// CODESYS_Control_for_Raspberry_Pi/Application/visualization/ups_s2/ups_s2_state
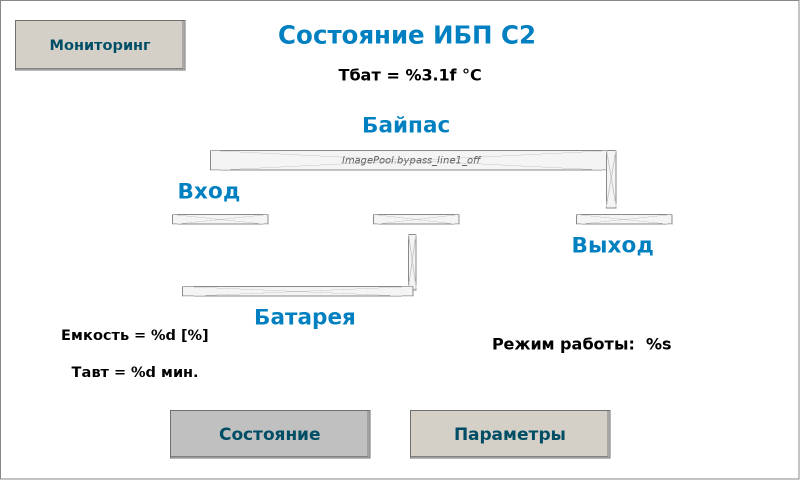
VISUALIZATION ups_s2_state  // 800x480, background image ImagePool.mpx_state_bg
    Rectangle (204,20 406x30), "Состояние ИБП С2"
    Button (410,410 200x48), "Параметры"
        OnMouseClick:  Assign=ups_s2_params, Type=Assignment
    Button (170,410 200x48), "Состояние", pressed state: PLC_PRG.var_true
    Rectangle (350,110 112x30), "Байпас"
    Rectangle (246,302 118x30), "Батарея"
    Rectangle (166,176 86x30), "Вход"
    Rectangle (560,230 106x30), "Выход"
    Rectangle (30,320 210x30), "Емкость = %d [%]", text variable: PLC_PRG.ips_s2_battery_capacity
    Rectangle (30,357 210x30), "Tавт = %d мин.", text variable: PLC_PRG.ips_s2_time_m
    Image (210,150 402x20), image: ImagePool.bypass_line1_off
        p84334746: PLC_PRG.ips_s2_bypass_line_state
    Image (606,150 10x58), image: ImagePool.bypass_arrow_off
        p84334746: PLC_PRG.ips_s2_bypass_arrow_state
    Image (576,214 96x10), image: ImagePool.arrow_off
        p84334746: PLC_PRG.ips_s2_output_state
    Image (172,214 96x10), image: ImagePool.arrow_off
        p84334746: PLC_PRG.ips_s2_input_state
    Image (408,234 8x56), image: ImagePool.battery_arrow_off
        p84334746: PLC_PRG.ips_s2_battery_arrow_state
    Image (182,286 231x10), image: ImagePool.battery_line_off
        p84334746: PLC_PRG.ips_s2_battery_line_state
    Button (15,20 170x50), "Мониторинг"
        OnMouseClick:  Assign=monitoring, Type=Assignment
    Rectangle (372,212 85x14)
    Image (373,214 86x10), image: ImagePool.arrow_off
        p84334746: PLC_PRG.ips_s2_arrow_state
    Rectangle (280,60 260x30), "Tбат = %3.1f °С", text variable: PLC_PRG.ips_s2_temp_real
    Rectangle (396,329 372x30), "Режим работы: %s", text variable: PLC_PRG.mpx_s2_state_string
    hotkey  Id=481037385728, Key=KeyDown=True, KeyName=0, VisuElemId=38
    hotkey  Id=481038434304, Key=KeyName=0, VisuElemId=38
END_VISUALIZATION

// CODESYS_Control_for_Raspberry_Pi/Application/visualization/main
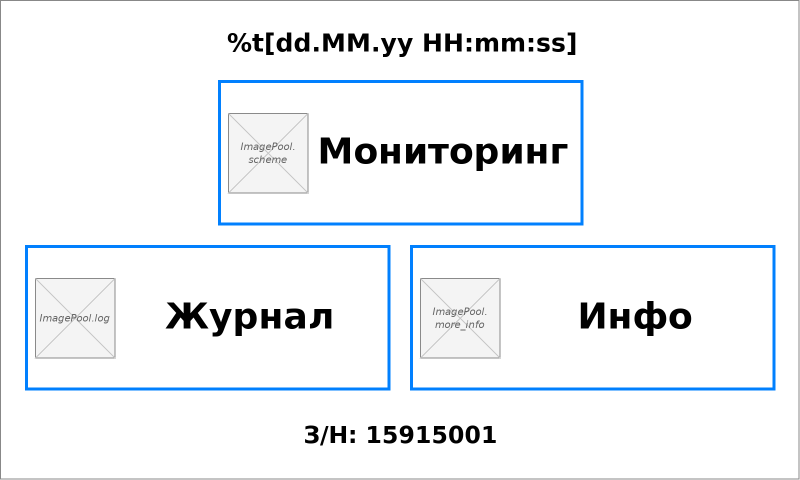
VISUALIZATION main  // 800x480, background image ImagePool.bg_800
    Group (218,80 365x145)
        OnMouseClick:  Assign=monitoring, Type=Assignment
        RoundedRectangle (0,0 365x145)
            OnMouseClick:  Assign=ups_s2_state, Type=Assignment
        RoundedRectangle (95,43 260x56), "Мониторинг"
        Image (10,33 80x80), image: ImagePool.scheme
    Group (25,245 365x145)
        OnMouseClick:  Assign=logs, Type=Assignment
        RoundedRectangle (0,0 365x145)
            OnMouseClick:  Assign=ups_s2_state, Type=Assignment
        RoundedRectangle (95,43 260x56), "Журнал"
            OnMouseClick:  Assign=ups_s2_state, Type=Assignment
        Image (10,33 80x80), image: ImagePool.log
    Group (410,245 365x145)
        OnMouseClick:  Assign=more, Type=Assignment
        RoundedRectangle (0,0 365x145)
            OnMouseClick:  Assign=ups_s2_state, Type=Assignment
        RoundedRectangle (95,43 260x56), "Инфо"
        Image (10,33 80x80), image: ImagePool.more_info
    Rectangle (215,20 375x45), "%t[dd.MM.yy HH:mm:ss]"
    Label (303,420 195x30), "З/Н: 15915001"
END_VISUALIZATION

// CODESYS_Control_for_Raspberry_Pi/Application/visualization/info
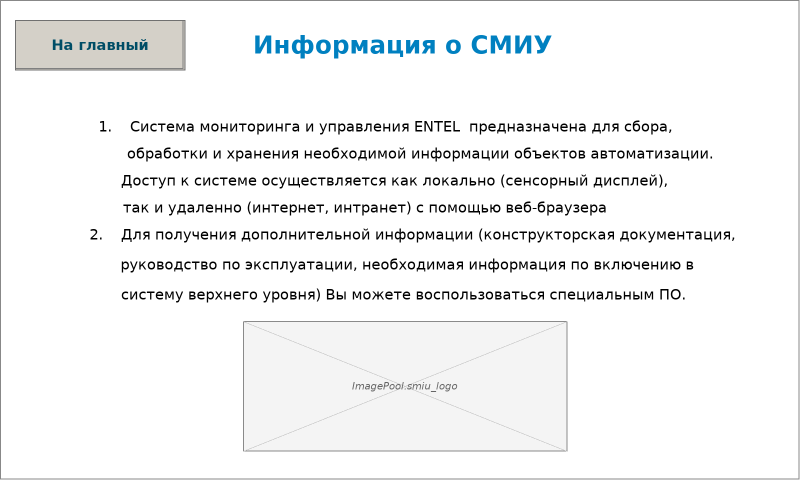
VISUALIZATION info  // 800x480, background image ImagePool.bg_800
    Rectangle (200,30 406x30), "Информация о СМИУ"
    Button (15,20 170x50), "На главный"
        OnMouseClick:  Assign=main, Type=Assignment
    Label (78,108 615x37), "1. Система мониторинга и управления ENTEL предназначена для сбора,"
    Label (120,135 601x37), "обработки и хранения необходимой информации объектов автоматизации."
    Label (99,162 591x37), "Доступ к системе осуществляется как локально (сенсорный дисплей),"
    Label (42,189 646x37), "так и удаленно (интернет, интранет) с помощью веб-браузера"
    Label (105,216 615x37), "2. Для получения дополнительной информации (конструкторская документация,"
    Label (120,243 601x37)
    Label (114,246 591x37), "руководство по эксплуатации, необходимая информация по включению в"
    Label (108,276 591x37), "систему верхнего уровня) Вы можете воспользоваться специальным ПО."
    Image (243,321 324x130), image: ImagePool.smiu_logo
END_VISUALIZATION

// CODESYS_Control_for_Raspberry_Pi/Application/visualization/climate
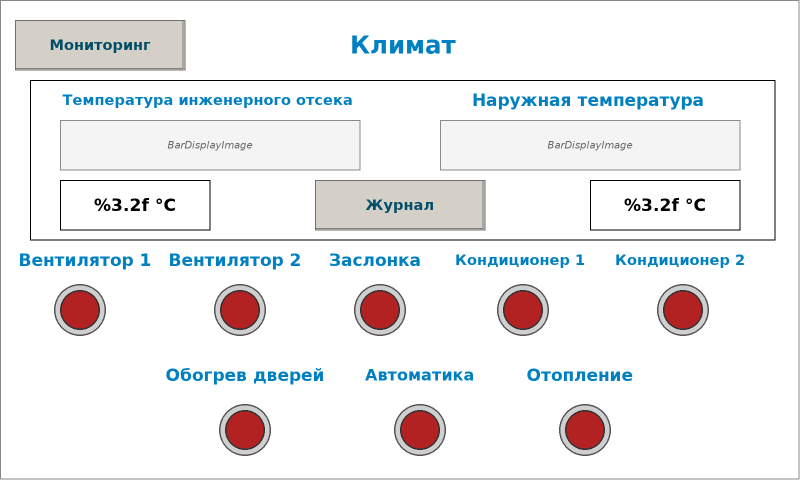
VISUALIZATION climate  // 800x480, background image ImagePool.bg_800
    Rectangle (200,30 406x30), "Климат"
    Button (15,20 170x50), "Мониторинг"
        OnMouseClick:  Assign=monitoring, Type=Assignment
    Rectangle (30,80 745x160)
    Rectangle (35,85 346x30), "Температура инженерного отсека"
    Rectangle (60,180 150x50), "%3.2f °С", text variable: PLC_PRG.climate_temp_in_real
    BarDisplayImage (60,120 300x50), value: PLC_PRG.climate_temp_in_real, style: BarDisplayImage-Gray, scale format: %.1f, scale -10..50
    Rectangle (415,85 346x30), "Наружная температура"
    Rectangle (590,180 150x50), "%3.2f °С", text variable: PLC_PRG.climate_temp_out_real
    BarDisplayImage (440,120 300x50), value: PLC_PRG.climate_temp_out_real, style: BarDisplayImage-Gray, scale format: %.1f, scale -60..80
    Rectangle (345,360 150x30), "Автоматика"
    Lamp1 (390,400 60x60), variable: PLC_PRG.climate_auto_state, style: Lamp-Lamp1-Red
    Lamp1 (50,280 60x60), variable: PLC_PRG.climate_vent_1_state, style: Lamp-Lamp1-Red
    Rectangle (10,250 150x20), "Вентилятор 1"
    Lamp1 (350,280 60x60), variable: PLC_PRG.climate_zaslonka_state, style: Lamp-Lamp1-Red
    Rectangle (320,250 110x20), "Заслонка"
    Rectangle (440,250 160x20), "Кондиционер 1"
    Lamp1 (490,280 66x60), variable: PLC_PRG.climate_condition_1_state, style: Lamp-Lamp1-Red
    Lamp1 (555,400 60x60), variable: PLC_PRG.climate_heat_state, style: Lamp-Lamp1-Red
    Rectangle (505,365 150x20), "Отопление"
    Lamp1 (210,280 60x60), variable: PLC_PRG.climate_vent_2_state, style: Lamp-Lamp1-Red
    Rectangle (160,250 150x20), "Вентилятор 2"
    Rectangle (600,250 160x20), "Кондиционер 2"
    Lamp1 (650,280 66x60), variable: PLC_PRG.climate_condition_2_state, style: Lamp-Lamp1-Red
    Lamp1 (215,400 60x60), variable: PLC_PRG.climate_heat_door_state, style: Lamp-Lamp1-Red
    Rectangle (155,365 180x20), "Обогрев дверей"
    Button (315,180 170x50), "Журнал"
        OnMouseClick:  Assign=climate_log, Type=Assignment
    hotkey  Id=481037385728, Key=KeyDown=True, KeyName=0, VisuElemId=3
    hotkey  Id=481038434304, Key=KeyName=0, VisuElemId=3
    hotkey  Id=481037385728, Key=KeyDown=True, KeyName=0, VisuElemId=73
    hotkey  Id=481038434304, Key=KeyName=0, VisuElemId=73
END_VISUALIZATION

// CODESYS_Control_for_Raspberry_Pi/Application/visualization/alarm
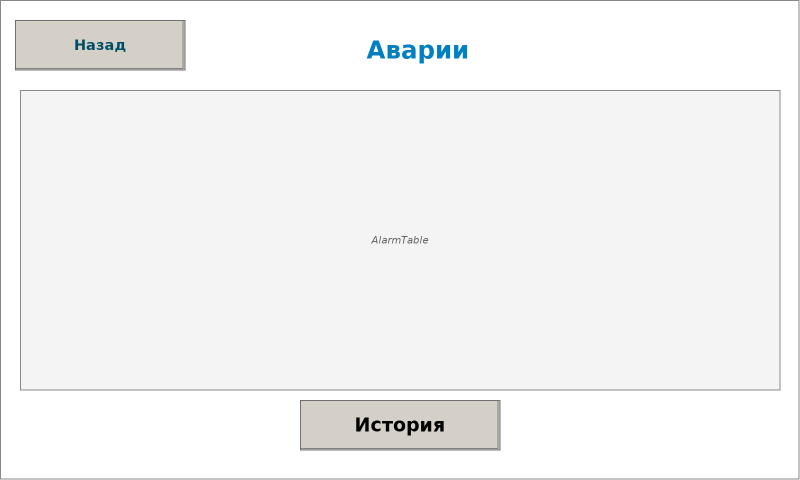
VISUALIZATION alarm  // 800x480, background image ImagePool.bg_800
    Button (300,400 200x50), "История", colour toggle: PLC_PRG.history
        toggle PLC_PRG.history
    Button (15,20 170x50), "Назад"
        OnMouseClick:  Assign=monitoring, Type=Previous
    AlarmTable (20,90 760x300)
        Column[0]: ColumnTitle=Временная отметка
        Column[1]: ColumnTitle=Сообщение
        p1521930926: AlarmGroup
        p1663851261: __All
        p3266827225: PLC_PRG.history
    Rectangle (215,35 406x30), "Аварии"
    hotkey  Id=481037385728, Key=KeyDown=True, KeyName=0, VisuElemId=6
    hotkey  Id=481038434304, Key=KeyName=0, VisuElemId=6
END_VISUALIZATION

// CODESYS_Control_for_Raspberry_Pi/Application/visualization/schrps
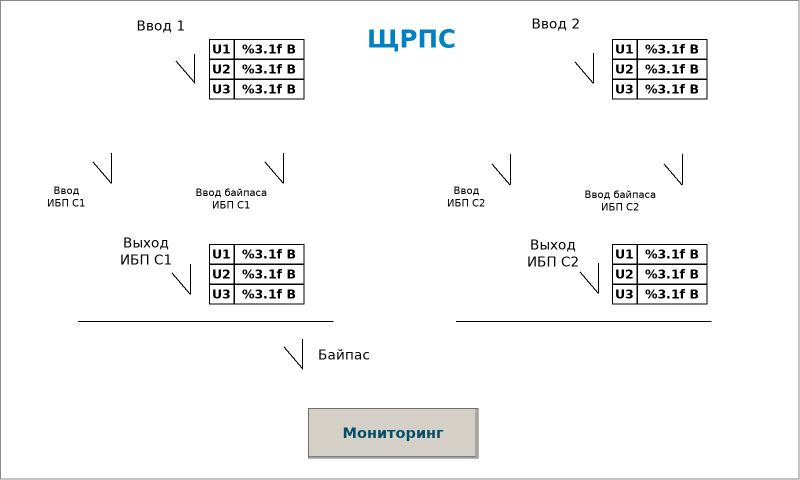
VISUALIZATION schrps  // 800x480, background image ImagePool.shrps
    Button (308,408 170x50), "Мониторинг"
        OnMouseClick:  Assign=monitoring, Type=Assignment
    Rectangle (316,24 191x30), "ЩРПC"
    Line (194,82) (176,61), invisible if: PLC_PRG.shrps_in_1
    Line (111,183) (93,162), invisible if: PLC_PRG.shrps_ups_in_1
    Line (283,183) (265,162), invisible if: PLC_PRG.shrps_bypass_in_1
    Line (190,294) (172,273), invisible if: PLC_PRG.shrps_ups_out_1
    Line (302,368) (284,347), invisible if: PLC_PRG.shrps_bypass_out
    Line (598,293) (580,272), invisible if: PLC_PRG.shrps_ups_out_2
    Line (510,185) (492,164), invisible if: PLC_PRG.shrps_ups_in_2
    Line (682,185) (664,164), invisible if: PLC_PRG.shrps_bypass_in_2
    Line (593,83) (575,62), invisible if: PLC_PRG.shrps_in_2
    Line (194,54) (194,83), invisible if: NOT(PLC_PRG.shrps_in_1)
    Line (283,153) (283,183), invisible if: NOT(PLC_PRG.shrps_bypass_in_1)
    Line (111,153) (111,183), invisible if: NOT(PLC_PRG.shrps_ups_in_1)
    Line (190,264) (190,294), invisible if: NOT(PLC_PRG.shrps_ups_out_1)
    Line (302,339) (302,369), invisible if: NOT(PLC_PRG.shrps_bypass_out)
    Line (598,263) (598,293), invisible if: NOT(PLC_PRG.shrps_ups_out_2)
    Line (682,154) (682,184), invisible if: NOT(PLC_PRG.shrps_bypass_in_2)
    Line (510,154) (510,184), invisible if: NOT(PLC_PRG.shrps_ups_in_2)
    Line (593,53) (593,83), invisible if: NOT(PLC_PRG.shrps_in_2)
    Label (317,340 54x30), "Байпас"
    Label (134,11 54x30), "Ввод 1"
    Label (529,9 54x30), "Ввод 2"
    Label (16,178 101x38), "Ввод ИБП С1"
    Label (416,178 101x38), "Ввод ИБП С2"
    Label (181,180 101x38), "Ввод байпаса ИБП С1"
    Label (570,182 101x38), "Ввод байпаса ИБП С2"
    Group (209,244 95x60)
        Rectangle (25,0 70x20), "%3.1f В", text variable: PLC_PRG.shrps_voltage_3_line_1
        Rectangle (0,0 25x20), "U1"
        Rectangle (0,20 25x20), "U2"
        Rectangle (25,20 70x20), "%3.1f В", text variable: PLC_PRG.shrps_voltage_3_line_2
        Rectangle (0,40 25x20), "U3"
        Rectangle (25,40 70x20), "%3.1f В", text variable: PLC_PRG.shrps_voltage_3_line_3
    Label (112,232 68x39), "Выход ИБП С1"
    Line (456,321) (711,321), colour toggle: PLC_PRG.shrps_ups_bus_2
    Line (78,321) (333,321), colour toggle: PLC_PRG.shrps_ups_bus_1
    Label (519,234 68x39), "Выход ИБП С2"
    Group (209,39 95x60)
        Rectangle (25,0 70x20), "%3.1f В", text variable: PLC_PRG.shrps_voltage_1_line_1
        Rectangle (0,0 25x20), "U1"
        Rectangle (0,20 25x20), "U2"
        Rectangle (25,20 70x20), "%3.1f В", text variable: PLC_PRG.shrps_voltage_1_line_2
        Rectangle (0,40 25x20), "U3"
        Rectangle (25,40 70x20), "%3.1f В", text variable: PLC_PRG.shrps_voltage_1_line_3
    Group (612,39 95x60)
        Rectangle (25,0 70x20), "%3.1f В", text variable: PLC_PRG.shrps_voltage_2_line_1
        Rectangle (0,0 25x20), "U1"
        Rectangle (0,20 25x20), "U2"
        Rectangle (25,20 70x20), "%3.1f В", text variable: PLC_PRG.shrps_voltage_2_line_2
        Rectangle (0,40 25x20), "U3"
        Rectangle (25,40 70x20), "%3.1f В", text variable: PLC_PRG.shrps_voltage_2_line_3
    Group (612,244 95x60)
        Rectangle (25,0 70x20), "%3.1f В", text variable: PLC_PRG.shrps_voltage_4_line_1
        Rectangle (0,0 25x20), "U1"
        Rectangle (0,20 25x20), "U2"
        Rectangle (25,20 70x20), "%3.1f В", text variable: PLC_PRG.shrps_voltage_4_line_2
        Rectangle (0,40 25x20), "U3"
        Rectangle (25,40 70x20), "%3.1f В", text variable: PLC_PRG.shrps_voltage_4_line_3
    hotkey  Id=481037385728, Key=KeyDown=True, KeyName=0, VisuElemId=1
    hotkey  Id=481038434304, Key=KeyName=0, VisuElemId=1
END_VISUALIZATION

// CODESYS_Control_for_Raspberry_Pi/Application/visualization/shasn
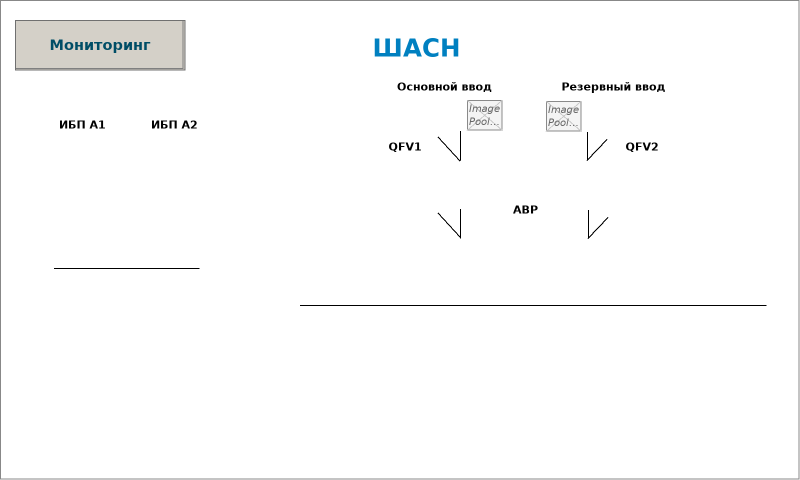
VISUALIZATION shasn  // 800x480, background image ImagePool.shasn
    Button (15,20 170x50), "Мониторинг"
        OnMouseClick:  Assign=monitoring, Type=Assignment
    Line (426,184)
    Line (460,237) (438,213), invisible if: GPIO_HANDLER.IN_9
    Line (460,209) (460,238), invisible if: NOT(GPIO_HANDLER.IN_9)
    Line (588,238) (608,217), invisible if: GPIO_HANDLER.IN_10
    Line (588,210) (588,238), invisible if: NOT(GPIO_HANDLER.IN_10)
    Line (300,305) (766,305), colour toggle: GPIO_HANDLER.IN_7
    Line (54,268) (199,268), colour toggle: GPIO_HANDLER.IN_6
    Image (467,100 35x30), invisible if: NOT(GPIO_HANDLER.IN_4), image: ImagePool.volt
    Line (664,184)
    Image (546,101 35x30), invisible if: NOT(GPIO_HANDLER.IN_5), image: ImagePool.volt
    Rectangle (321,33 191x30), "ШАСН"
    Line (460,161) (438,137), invisible if: GPIO_HANDLER.IN_11
    Line (460,131) (460,160), invisible if: NOT(GPIO_HANDLER.IN_11)
    Line (587,132) (587,160), invisible if: NOT(GPIO_HANDLER.IN_12)
    Line (587,160) (607,139), invisible if: GPIO_HANDLER.IN_12
    Label (52,110 61x30), "ИБП А1"
    Label (144,110 61x30), "ИБП А2"
    Label (390,72 109x30), "Основной ввод"
    Label (559,72 109x30), "Резервный ввод"
    Label (495,195 61x30), "АВР"
    Label (378,132 54x30), "QFV1"
    Label (615,132 54x30), "QFV2"
    hotkey  Id=481037385728, Key=KeyDown=True, KeyName=0, VisuElemId=1
    hotkey  Id=481038434304, Key=KeyName=0, VisuElemId=1
END_VISUALIZATION

// CODESYS_Control_for_Raspberry_Pi/Application/visualization/logs
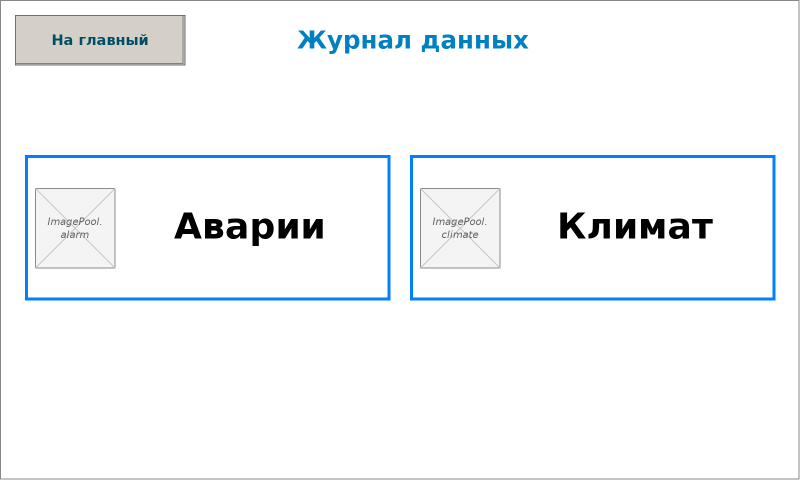
VISUALIZATION logs  // 800x480, background image ImagePool.bg_800
    Button (15,15 170x50), "На главный"
        OnMouseClick:  Assign=main, Type=Assignment
    Rectangle (210,25 406x30), "Журнал данных"
    Group (25,155 365x145)
        OnMouseClick:  Assign=alarm, Type=Assignment
        RoundedRectangle (0,0 365x145)
            OnMouseClick:  Assign=ups_s2_state, Type=Assignment
        RoundedRectangle (95,43 260x56), "Аварии"
        Image (10,33 80x80), image: ImagePool.alarm
    Group (410,155 365x145)
        OnMouseClick:  Assign=climate_log, Type=Assignment
        RoundedRectangle (0,0 365x145)
            OnMouseClick:  Assign=ups_s2_state, Type=Assignment
        RoundedRectangle (95,43 260x56), "Климат"
        Image (10,33 80x80), image: ImagePool.climate
    hotkey  Id=481037385728, Key=KeyDown=True, KeyName=0, VisuElemId=1
    hotkey  Id=481038434304, Key=KeyName=0, VisuElemId=1
END_VISUALIZATION

// CODESYS_Control_for_Raspberry_Pi/Application/visualization/schrpa
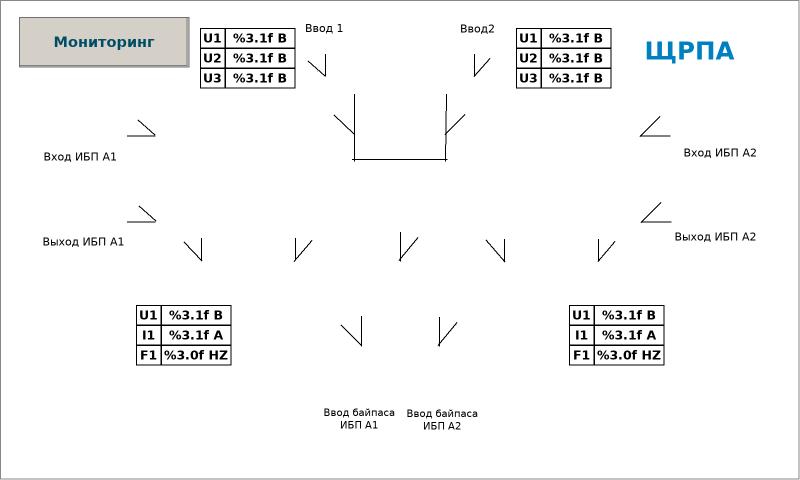
VISUALIZATION schrpa  // 800x480, background image ImagePool.shrpa_new
    Button (19,17 170x50), "Мониторинг"
        OnMouseClick:  Assign=monitoring, Type=Assignment
    Rectangle (594,36 191x30), "ЩРПА"
    Line (354,94) (354,161), invisible if: NOT(PLC_PRG.shrpa_input_switch_state_1)
    Line (354,134) (334,115), invisible if: PLC_PRG.shrpa_input_switch_state_1
    Line (352,159) (400,159), invisible if: NOT(PLC_PRG.shrpa_input_switch_state_1)
    Line (445,134) (465,114), invisible if: PLC_PRG.shrpa_input_switch_state_2
    Line (446,94) (445,161), invisible if: NOT(PLC_PRG.shrpa_input_switch_state_2)
    Line (399,159) (447,159), invisible if: NOT(PLC_PRG.shrpa_input_switch_state_2)
    Line (150,240)
    Line (202,261) (184,242), invisible if: PLC_PRG.shrpa_load_line_1_source_state_1
    Line (201,238) (201,260), invisible if: NOT(PLC_PRG.shrpa_load_line_1_source_state_1)
    Line (294,261) (312,240), invisible if: PLC_PRG.shrpa_load_line_1_source_state_2
    Line (295,238) (295,260), invisible if: NOT(PLC_PRG.shrpa_load_line_1_source_state_2)
    Line (487,239)
    Line (505,262) (486,240), invisible if: PLC_PRG.shrpa_load_line_2_source_state_1
    Line (504,239) (504,261), invisible if: NOT(PLC_PRG.shrpa_load_line_2_source_state_1)
    Line (598,261) (615,241), invisible if: PLC_PRG.shrpa_load_line_2_source_state_2
    Line (598,239) (598,261), invisible if: NOT(PLC_PRG.shrpa_load_line_2_source_state_2)
    Label (301,19 47x19), "Ввод 1"
    Label (453,19 49x20), "Ввод2"
    Label (27,142 107x30), "Вход ИБП А1"
    Label (667,138 107x30), "Вход ИБП А2"
    Label (30,227 107x30), "Выход ИБП А1"
    Label (662,222 107x30), "Выход ИБП А2"
    Label (309,400 101x38), "Ввод байпаса ИБП А1"
    Label (392,401 101x38), "Ввод байпаса ИБП А2"
    Line (640,136) (660,116), invisible if: PLC_PRG.shrpa_ups_in_2
    Line (474,76) (490,58), invisible if: PLC_PRG.shrpa_in_2
    Line (325,76) (308,61), invisible if: PLC_PRG.shrpa_in_1
    Line (155,135) (138,120), invisible if: PLC_PRG.shrpa_ups_in_1
    Line (361,345) (341,325), invisible if: PLC_PRG.shrpa_bypass_in_1
    Line (438,345) (457,322), invisible if: PLC_PRG.shrpa_bypass_in_2
    Line (361,316) (361,346), invisible if: NOT(PLC_PRG.shrpa_bypass_in_1)
    Line (439,317) (439,346), invisible if: NOT(PLC_PRG.shrpa_bypass_in_2)
    Line (670,136) (640,136), invisible if: NOT(PLC_PRG.shrpa_ups_in_2)
    Line (474,54) (474,76), invisible if: NOT(PLC_PRG.shrpa_in_2)
    Line (325,54) (325,76), invisible if: NOT(PLC_PRG.shrpa_in_1)
    Line (155,136) (127,136), invisible if: NOT(PLC_PRG.shrpa_ups_in_1)
    Line (317,71) (317,71)
    Line (156,221) (139,206), invisible if: PLC_PRG.shrpa_ups_out_1
    Line (155,222) (127,222), invisible if: NOT(PLC_PRG.shrpa_ups_out_1)
    Line (641,222) (661,202), invisible if: PLC_PRG.shrpa_ups_out_2
    Line (671,222) (641,222), invisible if: NOT(PLC_PRG.shrpa_ups_out_2)
    Line (400,232) (400,261), invisible if: NOT(PLC_PRG.shrpa_input_tv1)
    Line (399,260) (418,237), invisible if: PLC_PRG.shrpa_input_tv1
    Group (200,28 95x60)
        Rectangle (25,0 70x20), "%3.1f В", text variable: PLC_PRG.shrpa_voltage_1_line_1
        Rectangle (0,0 25x20), "U1"
        Rectangle (0,20 25x20), "U2"
        Rectangle (25,20 70x20), "%3.1f В", text variable: PLC_PRG.shrpa_voltage_1_line_2
        Rectangle (0,40 25x20), "U3"
        Rectangle (25,40 70x20), "%3.1f В", text variable: PLC_PRG.shrpa_voltage_1_line_3
    Group (516,28 95x60)
        Rectangle (25,0 70x20), "%3.1f В", text variable: PLC_PRG.shrpa_voltage_2_line_1
        Rectangle (0,0 25x20), "U1"
        Rectangle (0,20 25x20), "U2"
        Rectangle (25,20 70x20), "%3.1f В", text variable: PLC_PRG.shrpa_voltage_2_line_2
        Rectangle (0,40 25x20), "U3"
        Rectangle (25,40 70x20), "%3.1f В", text variable: PLC_PRG.shrpa_voltage_2_line_3
    Group (136,305 95x60)
        Rectangle (25,0 70x20), "%3.1f В", text variable: PLC_PRG.shrpa_voltage_3_line_1
        Rectangle (0,0 25x20), "U1"
        Rectangle (0,20 25x20), "I1"
        Rectangle (25,20 70x20), "%3.1f A", text variable: PLC_PRG.shrpa_current_3_line_1
        Rectangle (0,40 25x20), "F1"
        Rectangle (25,40 70x20), "%3.0f HZ", text variable: PLC_PRG.shrpa_freq_3_line_1
    Group (569,305 95x60)
        Rectangle (25,0 70x20), "%3.1f В", text variable: PLC_PRG.shrpa_voltage_4_line_1
        Rectangle (0,0 25x20), "U1"
        Rectangle (0,20 25x20), "I1"
        Rectangle (25,20 70x20), "%3.1f A", text variable: PLC_PRG.shrpa_current_4_line_1
        Rectangle (0,40 25x20), "F1"
        Rectangle (25,40 70x20), "%3.0f HZ", text variable: PLC_PRG.shrpa_freq_4_line_1
    hotkey  Id=481037385728, Key=KeyDown=True, KeyName=0, VisuElemId=1
    hotkey  Id=481038434304, Key=KeyName=0, VisuElemId=1
END_VISUALIZATION

// CODESYS_Control_for_Raspberry_Pi/Application/visualization/ups_s2/ups_s2_params
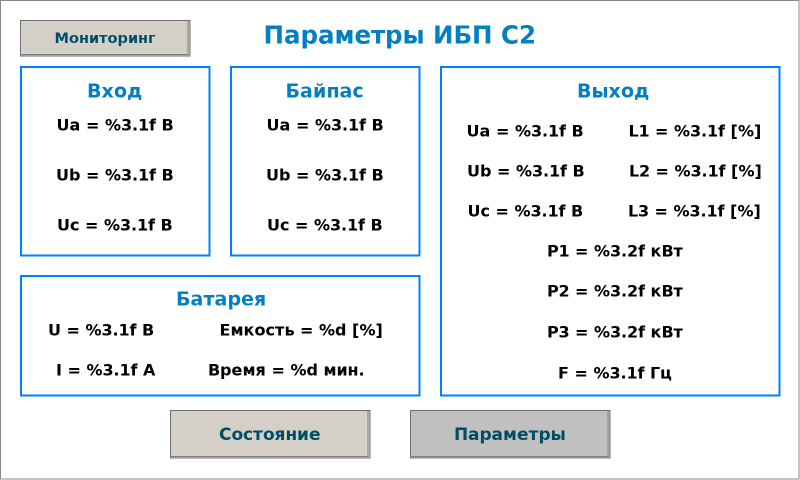
VISUALIZATION ups_s2_params  // 800x480, background image ImagePool.bg_800
    Rectangle (186,20 428x30), "Параметры ИБП С2"
    Button (170,410 200x48), "Состояние"
        OnMouseClick:  Assign=ups_s2_state, Type=Assignment
    Button (410,410 200x48), "Параметры", pressed state: PLC_PRG.var_true
    Button (20,20 170x36), "Мониторинг"
        OnMouseClick:  Assign=monitoring, Type=Assignment
    RoundedRectangle (440,66 340x330)
    RoundedRectangle (20,66 190x190)
    Rectangle (30,76 170x30), "Вход"
    Rectangle (25,110 180x30), "Ua = %3.1f В", text variable: PLC_PRG.ips_s2_in_v_1_real
    Rectangle (25,160 180x30), "Ub = %3.1f В", text variable: PLC_PRG.ips_s2_in_v_2_real
    Rectangle (25,210 180x30), "Uc = %3.1f В", text variable: PLC_PRG.ips_s2_in_v_3_real
    RoundedRectangle (230,66 190x190)
    Rectangle (240,76 170x30), "Байпас"
    Rectangle (235,110 180x30), "Ua = %3.1f В", text variable: PLC_PRG.ips_s2_bypass_v_1_real
    Rectangle (235,160 180x30), "Ub = %3.1f В", text variable: PLC_PRG.ips_s2_bypass_v_2_real
    Rectangle (235,210 180x30), "Uc = %3.1f В", text variable: PLC_PRG.ips_s2_bypass_v_3_real
    Rectangle (498,76 231x30), "Выход"
    Rectangle (446,116 158x30), "Ua = %3.1f В", text variable: PLC_PRG.ips_s2_output_v_1_real
    Rectangle (448,156 156x30), "Ub = %3.1f В", text variable: PLC_PRG.ips_s2_output_v_2_real
    Rectangle (447,196 157x30), "Uc = %3.1f В", text variable: PLC_PRG.ips_s2_output_v_3_real
    Rectangle (617,116 156x30), "L1 = %3.1f [%]", text variable: PLC_PRG.ips_s2_load_ph_1_real
    Rectangle (617,156 157x30), "L2 = %3.1f [%]", text variable: PLC_PRG.ips_s2_load_ph_2_real
    Rectangle (617,196 155x30), "L3 = %3.1f [%]", text variable: PLC_PRG.ips_s2_load_ph_3_real
    Rectangle (525,358 180x30), "F = %3.1f Гц", text variable: PLC_PRG.ips_s2_output_freq_real
    RoundedRectangle (20,275 400x121)
    Rectangle (30,290 382x18), "Батарея"
    Rectangle (26,315 150x30), "U = %3.1f В", text variable: PLC_PRG.ips_s2_battery_voltage_real
    Rectangle (31,355 150x30), "I = %3.1f A", text variable: PLC_PRG.ips_s2_battery_current_real
    Rectangle (189,315 225x30), "Емкость = %d [%]", text variable: PLC_PRG.ips_s2_battery_capacity
    Rectangle (525,236 180x30), "P1 = %3.2f кВт", text variable: PLC_PRG.ips_s2_output_active_power_1_real
    Rectangle (525,276 180x30), "P2 = %3.2f кВт", text variable: PLC_PRG.ips_s2_output_active_power_2_real
    Rectangle (525,317 180x30), "P3 = %3.2f кВт", text variable: PLC_PRG.ips_s2_output_active_power_3_real
    Rectangle (184,355 205x30), "Время = %d мин.", text variable: PLC_PRG.ips_s2_time_m
    hotkey  Id=481037385728, Key=KeyDown=True, KeyName=0, VisuElemId=7
    hotkey  Id=481038434304, Key=KeyName=0, VisuElemId=7
END_VISUALIZATION

// CODESYS_Control_for_Raspberry_Pi/Application/visualization/climate_log
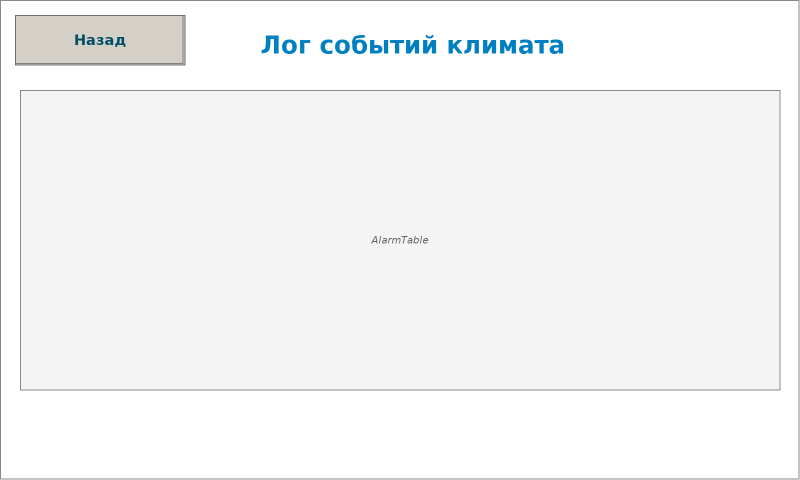
VISUALIZATION climate_log  // 800x480, background image ImagePool.bg_800
    Button (15,15 170x50), "Назад"
        OnMouseClick:  Assign=climate, Type=Previous
    Rectangle (210,30 406x30), "Лог событий климата"
    AlarmTable (20,90 760x300)
        Column[0]: ColumnTitle=Временная отметка
        Column[1]: ColumnTitle=Сообщение
        p1521930926: ClimateGroup
        p1663851261: __All
        p3266827225: PLC_PRG.var_true
    hotkey  Id=481037385728, Key=KeyDown=True, KeyName=0, VisuElemId=1
    hotkey  Id=481038434304, Key=KeyName=0, VisuElemId=1
END_VISUALIZATION

// CODESYS_Control_for_Raspberry_Pi/Application/visualization/more
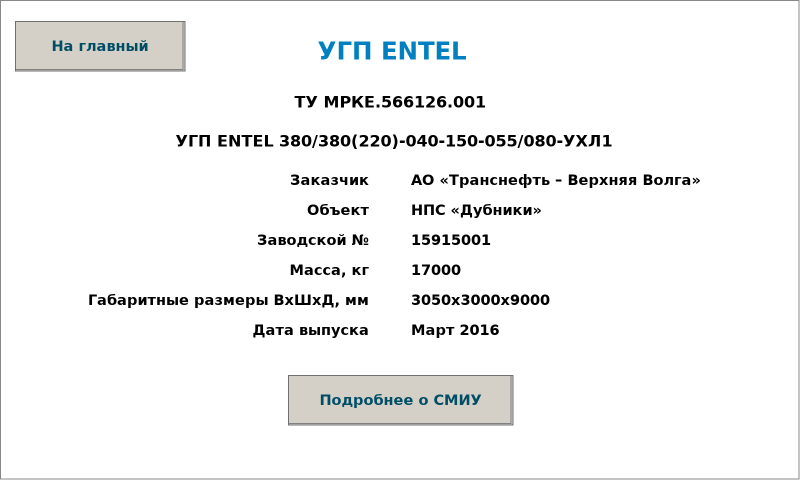
VISUALIZATION more  // 800x480, background image ImagePool.bg_800
    Rectangle (189,36 406x30), "УГП ENTEL"
    Button (15,21 170x50), "На главный"
        OnMouseClick:  Assign=main, Type=Assignment
    Button (288,375 225x50), "Подробнее о СМИУ"
        OnMouseClick:  Assign=info, Type=Assignment
    Label (213,87 355x30), "ТУ МРКЕ.566126.001"
    Label (191,126 406x30), "УГП ENTEL 380/380(220)-040-150-055/080-УХЛ1"
    Label (276,165 96x30), "Заказчик"
    Label (276,195 96x30), "Объект"
    Label (246,225 126x30), "Заводской №"
    Label (276,255 96x30), "Масса, кг"
    Label (96,285 276x30), "Габаритные размеры ВхШхД, мм"
    Label (201,315 171x30), "Дата выпуска"
    Label (408,165 309x30), "АО «Транснефть – Верхняя Волга»"
    Label (408,195 228x30), "НПС «Дубники»"
    Label (408,225 114x30), "15915001"
    Label (408,255 120x30), "17000"
    Label (408,285 165x30), "3050х3000х9000"
    Label (408,315 126x30), "Март 2016"
    hotkey  Id=481037385728, Key=KeyDown=True, KeyName=0, VisuElemId=3
    hotkey  Id=481038434304, Key=KeyName=0, VisuElemId=3
    hotkey  Id=481037385728, Key=KeyDown=True, KeyName=0, VisuElemId=5
    hotkey  Id=481038434304, Key=KeyName=0, VisuElemId=5
END_VISUALIZATION

// CODESYS_Control_for_Raspberry_Pi/Application/visualization/ups_s1/ups_s1_params
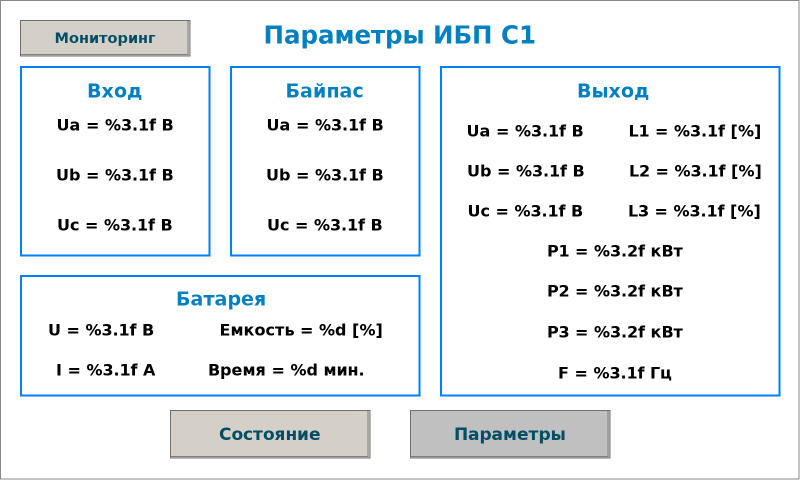
VISUALIZATION ups_s1_params  // 800x480, background image ImagePool.bg_800
    Rectangle (186,20 428x30), "Параметры ИБП С1"
    Button (170,410 200x48), "Состояние"
        OnMouseClick:  Assign=ups_s1_state, Type=Assignment
    Button (410,410 200x48), "Параметры", pressed state: PLC_PRG.var_true
    Button (20,20 170x36), "Мониторинг"
        OnMouseClick:  Assign=monitoring, Type=Assignment
    RoundedRectangle (440,66 340x330)
    RoundedRectangle (20,66 190x190)
    Rectangle (30,76 170x30), "Вход"
    Rectangle (25,110 180x30), "Ua = %3.1f В", text variable: PLC_PRG.ips_s1_in_v_1_real
    Rectangle (25,160 180x30), "Ub = %3.1f В", text variable: PLC_PRG.ips_s1_in_v_2_real
    Rectangle (25,210 180x30), "Uc = %3.1f В", text variable: PLC_PRG.ips_s1_in_v_3_real
    RoundedRectangle (230,66 190x190)
    Rectangle (240,76 170x30), "Байпас"
    Rectangle (235,110 180x30), "Ua = %3.1f В", text variable: PLC_PRG.ips_s1_bypass_v_1_real
    Rectangle (235,160 180x30), "Ub = %3.1f В", text variable: PLC_PRG.ips_s1_bypass_v_2_real
    Rectangle (235,210 180x30), "Uc = %3.1f В", text variable: PLC_PRG.ips_s1_bypass_v_3_real
    Rectangle (498,76 231x30), "Выход"
    Rectangle (446,116 158x30), "Ua = %3.1f В", text variable: PLC_PRG.ips_s1_output_v_1_real
    Rectangle (448,156 156x30), "Ub = %3.1f В", text variable: PLC_PRG.ips_s1_output_v_2_real
    Rectangle (447,196 157x30), "Uc = %3.1f В", text variable: PLC_PRG.ips_s1_output_v_3_real
    Rectangle (617,116 156x30), "L1 = %3.1f [%]", text variable: PLC_PRG.ips_s1_load_ph_1_real
    Rectangle (617,156 157x30), "L2 = %3.1f [%]", text variable: PLC_PRG.ips_s1_load_ph_2_real
    Rectangle (617,196 155x30), "L3 = %3.1f [%]", text variable: PLC_PRG.ips_s1_load_ph_3_real
    Rectangle (525,358 180x30), "F = %3.1f Гц", text variable: PLC_PRG.ips_s1_output_freq_real
    RoundedRectangle (20,275 400x121)
    Rectangle (30,290 382x18), "Батарея"
    Rectangle (26,315 150x30), "U = %3.1f В", text variable: PLC_PRG.ips_s1_battery_voltage_real
    Rectangle (31,355 150x30), "I = %3.1f A", text variable: PLC_PRG.ips_s1_battery_current_real
    Rectangle (189,315 225x30), "Емкость = %d [%]", text variable: PLC_PRG.ips_s1_battery_capacity
    Rectangle (525,236 180x30), "P1 = %3.2f кВт", text variable: PLC_PRG.ips_s1_output_active_power_1_real
    Rectangle (525,276 180x30), "P2 = %3.2f кВт", text variable: PLC_PRG.ips_s1_output_active_power_2_real
    Rectangle (525,317 180x30), "P3 = %3.2f кВт", text variable: PLC_PRG.ips_s1_output_active_power_3_real
    Rectangle (184,355 205x30), "Время = %d мин.", text variable: PLC_PRG.ips_s1_time_m
    hotkey  Id=481037385728, Key=KeyDown=True, KeyName=0, VisuElemId=7
    hotkey  Id=481038434304, Key=KeyName=0, VisuElemId=7
END_VISUALIZATION

// CODESYS_Control_for_Raspberry_Pi/Application/visualization/ups_a1/ups_a1_params
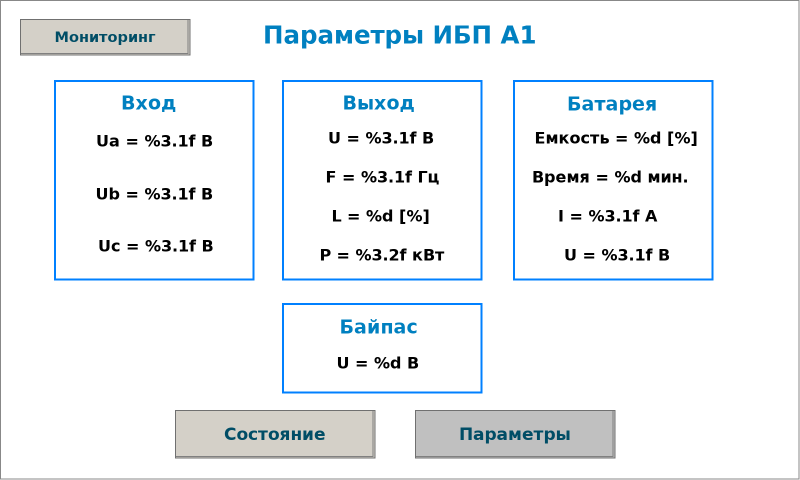
VISUALIZATION ups_a1_params  // 800x480, background image ImagePool.bg_800
    RoundedRectangle (513,80 200x200)
    Rectangle (186,20 428x30), "Параметры ИБП А1"
    Button (175,410 200x48), "Состояние"
        OnMouseClick:  Assign=ups_a1_state, Type=Assignment
    Button (415,410 200x48), "Параметры", pressed state: PLC_PRG.var_true
    Button (20,19 170x36), "Мониторинг"
        OnMouseClick:  Assign=monitoring, Type=Assignment
    RoundedRectangle (54,80 200x200)
    Rectangle (64,88 170x30), "Вход"
    Rectangle (60,126 189x30), "Ua = %3.1f В", text variable: PLC_PRG.ips_a1_in_v_1_real
    Rectangle (63,179 183x30), "Ub = %3.1f В", text variable: PLC_PRG.ips_a1_in_v_2_real
    Rectangle (63,231 186x30), "Uc = %3.1f В", text variable: PLC_PRG.ips_a1_in_v_3_real
    RoundedRectangle (282,303 200x90)
    Rectangle (294,312 170x30), "Байпас"
    Rectangle (303,348 150x30), "U = %d В", text variable: PLC_PRG.ips_a1_bypass_v_1_real
    RoundedRectangle (282,80 200x200)
    Rectangle (302,88 154x30), "Выход"
    Rectangle (291,123 180x30), "U = %3.1f В", text variable: PLC_PRG.ips_a1_output_v_1_real
    Rectangle (288,201 186x30), "L = %d [%]", text variable: PLC_PRG.ips_a1_load_ph_1_real
    Rectangle (302,240 160x30), "P = %3.2f кВт", text variable: PLC_PRG.ips_a1_output_active_power_1_real
    Rectangle (291,162 183x30), "F = %3.1f Гц", text variable: PLC_PRG.ips_a1_output_freq_real
    Rectangle (531,89 162x30), "Батарея"
    Rectangle (537,240 160x30), "U = %3.1f В", text variable: PLC_PRG.ips_a1_battery_voltage_real
    Rectangle (528,201 160x30), "I = %3.1f A", text variable: PLC_PRG.ips_a1_battery_current_real
    Rectangle (522,123 189x30), "Емкость = %d [%]", text variable: PLC_PRG.ips_a1_battery_capacity
    Rectangle (516,162 189x30), "Время = %d мин.", text variable: PLC_PRG.ips_a1_time_m
    hotkey  Id=481037385728, Key=KeyDown=True, KeyName=0, VisuElemId=7
    hotkey  Id=481038434304, Key=KeyName=0, VisuElemId=7
END_VISUALIZATION

// CODESYS_Control_for_Raspberry_Pi/Application/visualization/ups_s1/ups_s1_state
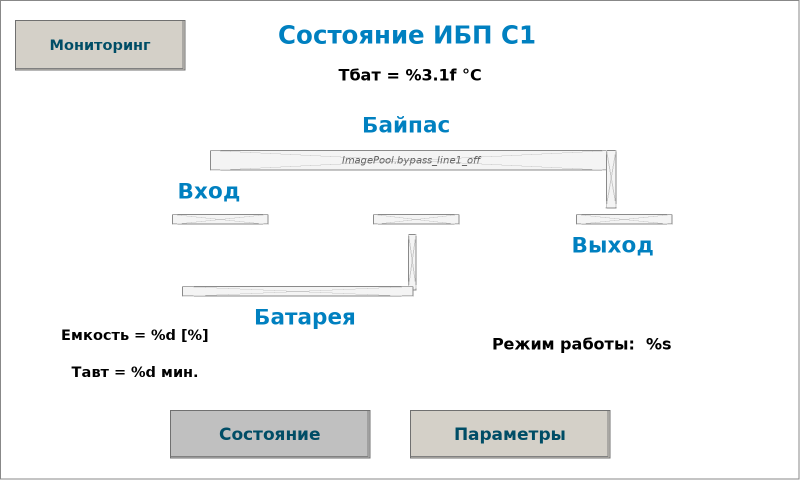
VISUALIZATION ups_s1_state  // 800x480, background image ImagePool.mpx_state_bg
    Rectangle (204,20 406x30), "Состояние ИБП С1"
    Button (410,410 200x48), "Параметры"
        OnMouseClick:  Assign=ups_s1_params, Type=Assignment
    Button (170,410 200x48), "Состояние", pressed state: PLC_PRG.var_true
    Rectangle (350,110 112x30), "Байпас"
    Rectangle (246,302 118x30), "Батарея"
    Rectangle (166,176 86x30), "Вход"
    Rectangle (560,230 106x30), "Выход"
    Rectangle (280,60 260x30), "Tбат = %3.1f °С", text variable: PLC_PRG.ips_s1_temp_real
    Rectangle (30,320 210x30), "Емкость = %d [%]", text variable: PLC_PRG.ips_s1_battery_capacity
    Rectangle (30,357 210x30), "Tавт = %d мин.", text variable: PLC_PRG.ips_s1_time_m
    Image (210,150 402x20), image: ImagePool.bypass_line1_off
        p84334746: PLC_PRG.ips_s1_bypass_line_state
    Image (606,150 10x58), image: ImagePool.bypass_arrow_off
        p84334746: PLC_PRG.ips_s1_bypass_arrow_state
    Image (576,214 96x10), image: ImagePool.arrow_off
        p84334746: PLC_PRG.ips_s1_output_state
    Image (172,214 96x10), image: ImagePool.arrow_off
        p84334746: PLC_PRG.ips_s1_input_state
    Image (408,234 8x56), image: ImagePool.battery_arrow_off
        p84334746: PLC_PRG.ips_s1_battery_arrow_state
    Image (182,286 231x10), image: ImagePool.battery_line_off
        p84334746: PLC_PRG.ips_s1_battery_line_state
    Button (15,20 170x50), "Мониторинг"
        OnMouseClick:  Assign=monitoring, Type=Assignment
    Rectangle (372,212 85x14)
    Image (373,214 86x10), image: ImagePool.arrow_off
        p84334746: PLC_PRG.ips_s1_arrow_state
    Rectangle (396,329 372x30), "Режим работы: %s", text variable: PLC_PRG.mpx_s1_state_string
    hotkey  Id=481037385728, Key=KeyDown=True, KeyName=0, VisuElemId=38
    hotkey  Id=481038434304, Key=KeyName=0, VisuElemId=38
END_VISUALIZATION

// CODESYS_Control_for_Raspberry_Pi/Application/visualization/ups_a2/ups_a2_state
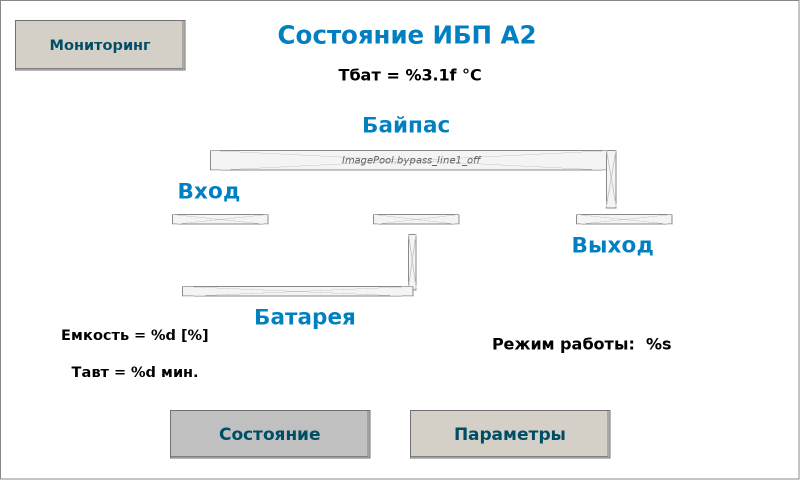
VISUALIZATION ups_a2_state  // 800x480, background image ImagePool.mpx_state_bg
    Rectangle (204,20 406x30), "Состояние ИБП А2"
    Button (410,410 200x48), "Параметры"
        OnMouseClick:  Assign=ups_a2_params, Type=Assignment
    Button (170,410 200x48), "Состояние", pressed state: PLC_PRG.var_true
    Rectangle (350,110 112x30), "Байпас"
    Rectangle (246,302 118x30), "Батарея"
    Rectangle (166,176 86x30), "Вход"
    Rectangle (560,230 106x30), "Выход"
    Rectangle (30,320 210x30), "Емкость = %d [%]", text variable: PLC_PRG.ips_a2_battery_capacity
    Rectangle (30,357 210x30), "Tавт = %d мин.", text variable: PLC_PRG.ips_a2_time_m
    Image (210,150 402x20), image: ImagePool.bypass_line1_off
        p84334746: PLC_PRG.ips_a2_bypass_line_state
    Image (606,150 10x58), image: ImagePool.bypass_arrow_off
        p84334746: PLC_PRG.ips_a2_bypass_arrow_state
    Image (576,214 96x10), image: ImagePool.arrow_off
        p84334746: PLC_PRG.ips_a2_output_state
    Image (172,214 96x10), image: ImagePool.arrow_off
        p84334746: PLC_PRG.ips_a2_input_state
    Image (408,234 8x56), image: ImagePool.battery_arrow_off
        p84334746: PLC_PRG.ips_a2_battery_arrow_state
    Image (182,286 231x10), image: ImagePool.battery_line_off
        p84334746: PLC_PRG.ips_a2_battery_line_state
    Button (15,20 170x50), "Мониторинг"
        OnMouseClick:  Assign=monitoring, Type=Assignment
    Rectangle (372,212 85x14)
    Image (373,214 86x10), image: ImagePool.arrow_off
        p84334746: PLC_PRG.ips_a2_arrow_state
    Rectangle (280,60 260x30), "Tбат = %3.1f °С", text variable: PLC_PRG.ips_a2_temp_real
    Rectangle (396,329 372x30), "Режим работы: %s", text variable: PLC_PRG.mpx_a2_state_string
    hotkey  Id=481037385728, Key=KeyDown=True, KeyName=0, VisuElemId=38
    hotkey  Id=481038434304, Key=KeyName=0, VisuElemId=38
END_VISUALIZATION

// CODESYS_Control_for_Raspberry_Pi/Application/visualization/ups_a1/ups_a1_state
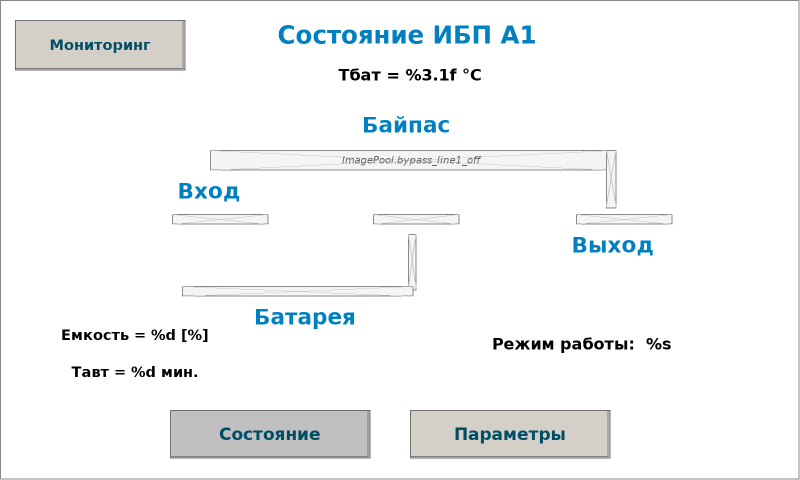
VISUALIZATION ups_a1_state  // 800x480, background image ImagePool.mpx_state_bg
    Rectangle (204,20 406x30), "Состояние ИБП А1"
    Button (410,410 200x48), "Параметры"
        OnMouseClick:  Assign=ups_a1_params, Type=Assignment
    Button (170,410 200x48), "Состояние", pressed state: PLC_PRG.var_true
    Rectangle (350,110 112x30), "Байпас"
    Rectangle (246,302 118x30), "Батарея"
    Rectangle (166,176 86x30), "Вход"
    Rectangle (560,230 106x30), "Выход"
    Rectangle (30,320 210x30), "Емкость = %d [%]", text variable: PLC_PRG.ips_a1_battery_capacity
    Rectangle (30,357 210x30), "Tавт = %d мин.", text variable: PLC_PRG.ips_a1_time_m
    Image (210,150 402x20), image: ImagePool.bypass_line1_off
        p84334746: PLC_PRG.ips_a1_bypass_line_state
    Image (606,150 10x58), image: ImagePool.bypass_arrow_off
        p84334746: PLC_PRG.ips_a1_bypass_arrow_state
    Image (576,214 96x10), image: ImagePool.arrow_off
        p84334746: PLC_PRG.ips_a1_output_state
    Image (172,214 96x10), image: ImagePool.arrow_off
        p84334746: PLC_PRG.ips_a1_input_state
    Image (408,234 8x56), image: ImagePool.battery_arrow_off
        p84334746: PLC_PRG.ips_a1_battery_arrow_state
    Image (182,286 231x10), image: ImagePool.battery_line_off
        p84334746: PLC_PRG.ips_a1_battery_line_state
    Button (15,20 170x50), "Мониторинг"
        OnMouseClick:  Assign=monitoring, Type=Assignment
    Rectangle (372,212 85x14)
    Image (373,214 86x10), image: ImagePool.arrow_off
        p84334746: PLC_PRG.ips_a1_arrow_state
    Rectangle (280,60 260x30), "Tбат = %3.1f °С", text variable: PLC_PRG.ips_a1_temp_real
    Rectangle (396,329 372x30), "Режим работы: %s", text variable: PLC_PRG.mpx_a1_state_string
    hotkey  Id=481037385728, Key=KeyDown=True, KeyName=0, VisuElemId=38
    hotkey  Id=481038434304, Key=KeyName=0, VisuElemId=38
END_VISUALIZATION

// CODESYS_Control_for_Raspberry_Pi/Application/visualization/ups_a2/ups_a2_params
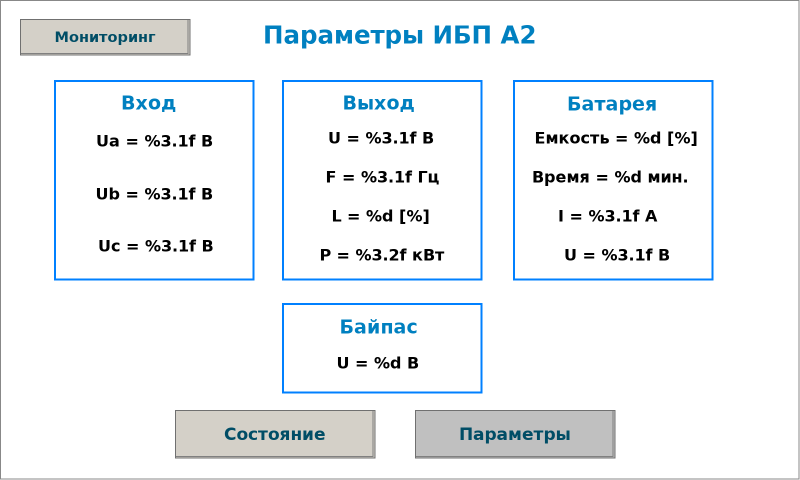
VISUALIZATION ups_a2_params  // 800x480, background image ImagePool.bg_800
    RoundedRectangle (513,80 200x200)
    Rectangle (186,20 428x30), "Параметры ИБП А2"
    Button (175,410 200x48), "Состояние"
        OnMouseClick:  Assign=ups_a2_state, Type=Assignment
    Button (415,410 200x48), "Параметры", pressed state: PLC_PRG.var_true
    Button (20,19 170x36), "Мониторинг"
        OnMouseClick:  Assign=monitoring, Type=Assignment
    RoundedRectangle (54,80 200x200)
    Rectangle (64,88 170x30), "Вход"
    Rectangle (60,126 189x30), "Ua = %3.1f В", text variable: PLC_PRG.ips_a2_in_v_1_real
    Rectangle (63,179 183x30), "Ub = %3.1f В", text variable: PLC_PRG.ips_a2_in_v_2_real
    Rectangle (63,231 186x30), "Uc = %3.1f В", text variable: PLC_PRG.ips_a2_in_v_3_real
    RoundedRectangle (282,303 200x90)
    Rectangle (294,312 170x30), "Байпас"
    Rectangle (303,348 150x30), "U = %d В", text variable: PLC_PRG.ips_a2_bypass_v_1_real
    RoundedRectangle (282,80 200x200)
    Rectangle (302,88 154x30), "Выход"
    Rectangle (291,123 180x30), "U = %3.1f В", text variable: PLC_PRG.ips_a2_output_v_1_real
    Rectangle (288,201 186x30), "L = %d [%]", text variable: PLC_PRG.ips_a2_load_ph_1_real
    Rectangle (302,240 160x30), "P = %3.2f кВт", text variable: PLC_PRG.ips_a2_output_active_power_1_real
    Rectangle (291,162 183x30), "F = %3.1f Гц", text variable: PLC_PRG.ips_a2_output_freq_real
    Rectangle (531,89 162x30), "Батарея"
    Rectangle (537,240 160x30), "U = %3.1f В", text variable: PLC_PRG.ips_a2_battery_voltage_real
    Rectangle (528,201 160x30), "I = %3.1f A", text variable: PLC_PRG.ips_a2_battery_current_real
    Rectangle (522,123 189x30), "Емкость = %d [%]", text variable: PLC_PRG.ips_a2_battery_capacity
    Rectangle (516,162 189x30), "Время = %d мин.", text variable: PLC_PRG.ips_a2_time_m
    hotkey  Id=481037385728, Key=KeyDown=True, KeyName=0, VisuElemId=7
    hotkey  Id=481038434304, Key=KeyName=0, VisuElemId=7
END_VISUALIZATION

(* text list AlarmGroup (id | default)
  103 | ИБП С2 работает от АКБ
  102 | ИБП С1 работает от АКБ
  101 | Отсутствует напряжение на резервном вводе ЩРПС
  100 | Отсутствует напряжение на основном вводе ЩРПC
  99 | Отсутствует напряжение на ШБПА  ЩРПА
  98 | Авария ШОС
  97 | Нарушение ШОС
  96 | Пожар
  95 | Отсутствует напряжение на выходе ИБП А2
  94 | Отсутствует напряжение на выходе ИБП А1
  93 | Отсутствует напряжение на выходе ИБП С2
  92 | Отсутствует напряжение на выходе ИБП С1
  91 | Отсутствует напряжение на входе ИБП А2
  90 | Отсутствует напряжение на входе ИБП А1
  89 | Отсутствует напряжение на входе ИБП С2
  88 | Отсутствует напряжение на входе ИБП С1
  87 | Включен ручной режим байпас ИБП А2
  86 | Отсутствует напряжения на выходе ИБПС 2 модуль 4 (1ф.)
  85 | Включен ручной режим байпас ИБП А1
  84 | Отсутствует напряжения на выходе ИБПС 2 модуль 4 (3ф.)
  83 | Отсутствует напряжения на выходе ИБПС 2 модуль 4 (2ф.)
  82 | Отсутствует напряжения на выходе ИБПС 2 модуль 4 (1ф.)
  81 | Отсутствует напряжения на выходе ИБПС 2 модуль 3 (3ф.)
  80 | Отсутствует напряжения на выходе ИБПС 2 модуль 3 (2ф.)
  79 | Отсутствует напряжения на выходе ИБПС 2 модуль 3 (1ф.)
  78 | Отсутствует напряжения на выходе ИБПС 2 модуль 2 (3ф.)
  77 | Отсутствует напряжения на выходе ИБПС 2 модуль 2 (2ф.)
  76 | Отсутствует напряжения на выходе ИБПС 2 модуль 2 (1ф.)
  75 | Отсутствует напряжения на выходе ИБПС 2 модуль 1 (3ф.)
  74 | Отсутствует напряжения на выходе ИБПС 2 модуль 1 (2ф.)
  73 | Отсутствует напряжения на выходе ИБПС 2 модуль 1 (1ф.)
  72 | Отсутствует напряжения на выходе ИБПС 1 модуль 4 (3ф.)
  71 | Отсутствует напряжения на выходе ИБПС 1 модуль 4 (2ф.)
  70 | Отсутствует напряжения на выходе ИБПС 1 модуль 4 (1ф.)
  69 | Отсутствует напряжения на выходе ИБПС 1 модуль 3 (3ф.)
  68 | Отсутствует напряжения на выходе ИБПС 1 модуль 3 (2ф.)
  67 | Отсутствует напряжения на выходе ИБПС 1 модуль 3 (1ф.)
  66 | Отсутствует напряжения на выходе ИБПС 1 модуль 2 (3ф.)
  65 | Отсутствует напряжения на выходе ИБПС 1 модуль 2 (2ф.)
  64 | Отсутствует напряжения на выходе ИБПС 1 модуль 2 (1ф.)
  63 | Отсутствует напряжения на выходе ИБПС 1 модуль 1 (3ф.)
  62 | Отсутствует напряжения на выходе ИБПС 1 модуль 1 (2ф.)
  61 | Отсутствует напряжения на выходе ИБПС 1 модуль 1 (1ф.)
  60 | Отсутствует напряжения на выходе ИБПА 2 модуль 2
  59 | Отсутствует напряжения на выходе ИБПА 2 модуль 1
  58 | Отсутствует напряжения на выходе ИБПА 1 модуль 2
  57 | Отсутствует напряжения на выходе ИБПА 1 модуль 1
  56 | Авария ИБПС 2 модуль 4
  55 | Авария ИБПС 2 модуль 3
  54 | Авария ИБПС 2 модуль 2
  53 | Авария ИБП С2
  52 | Авария ИБПС 1 модуль 4
  51 | Авария ИБПС 1 модуль 3
  50 | Авария ИБПС 1 модуль 2
  49 | Авария ИБП С1
  48 | Авария ИБПА 2 модуль 2
  47 | Авария ИБП А2
  46 | Авария ИБПА 1 модуль 2
  45 | Авария ИБП А1
  44 | Отсутствует напряжение на входе ИБПC 2 модуль 4 (3 ф.)
  43 | Отсутствует напряжение на входе ИБПC 2 модуль 4 (2 ф.)
  42 | Отсутствует напряжение на входе ИБПC 2 модуль 4 (1 ф.)
  41 | Отсутствует напряжение на входе ИБПC 2 модуль 3 (3 ф.)
  40 | Отсутствует напряжение на входе ИБПC 2 модуль 3 (2 ф.)
  39 | Отсутствует напряжение на входе ИБПC 2 модуль 3 (1 ф.)
  38 | Отсутствует напряжение на входе ИБПC 2 модуль 2 (3 ф.)
  37 | Отсутствует напряжение на входе ИБПC 2 модуль 2 (2 ф.)
  36 | Отсутствует напряжение на входе ИБПC 2 модуль 2 (1 ф.)
  35 | Отсутствует напряжение на входе ИБПC 2 модуль 1 (3 ф.)
  34 | Отсутствует напряжение на входе ИБПC 2 модуль 1 (2 ф.)
  33 | Отсутствует напряжение на входе ИБПC 2 модуль 1 (1 ф.)
  32 | Отсутствует напряжение на входе ИБПC 1 модуль 4 (3 ф.)
  31 | Отсутствует напряжение на входе ИБПC 1 модуль 4 (2 ф.)
  30 | Отсутствует напряжение на входе ИБПC 1 модуль 4 (1 ф.)
  29 | Отсутствует напряжение на входе ИБПC 1 модуль 3 (3 ф.)
  28 | Отсутствует напряжение на входе ИБПC 1 модуль 3 (2 ф.)
  27 | Отсутствует напряжение на входе ИБПC 1 модуль 3 (1 ф.)
  26 | Отсутствует напряжение на входе ИБПC 1 модуль 2 (3 ф.)
  25 | Отсутствует напряжение на входе ИБПC 1 модуль 2 (2 ф.)
  24 | Отсутствует напряжение на входе ИБПC 1 модуль 1 (3 ф.)
  23 | Отсутствует напряжение на входе ИБПC 1 модуль 2 (1 ф.)
  22 | Отсутствует напряжение на входе ИБПC 1 модуль 1 (2 ф.)
  21 | Отсутствует напряжение на входе ИБПC 1 модуль 1 (1 ф.)
  20 | Отсутствует напряжение на входе ИБПА 2 модуль 2 (3 ф.)
  19 | Отсутствует напряжение на входе ИБПА 2 модуль 2 (2 ф.)
  18 | Отсутствует напряжение на входе ИБПА 2 модуль 2 (1 ф.)
  17 | Отсутствует напряжение на входе ИБПА 2 модуль 1 (3 ф.)
  16 | Отсутствует напряжение на входе ИБПА 2 модуль 1 (2 ф.)
  15 | Отсутствует напряжение на входе ИБПА 2 модуль 1 (1 ф.)
  14 | Отсутствует напряжение на входе ИБПА 1 модуль 2 (3 ф.)
  13 | Отсутствует напряжение на входе ИБПА 1 модуль 2 (2 ф.)
  12 | Отсутствует напряжение на входе ИБПА 1 модуль 2 (1 ф.)
  11 | Отсутствует напряжение на входе ИБПА 1 модуль 1 (3 ф.)
  10 | Отсутствует напряжение на входе ИБПА 1 модуль 1 (2 ф.)
  9 | 
  8 | Отсутствует напряжение на входе ИБПА 1 модуль 1 (1 ф.)
  7 | Отсутствует напряжение на шине ГП ШАСН
  6 | Отсутствует напряжение на шине БП ШАСН
  5 | Отсутствует напряжение на ГП 2 ЩРПС
  4 | Отсутствует напряжение на ГП 1 ЩРПС
  3 | Отсутствует напряжение на резервном вводе ШАСН
  2 | Отсутствует напряжение на основном вводе ШАСН
  1 | Отсутствует напряжение на резервном вводе ЩРПА
  0 | Отсутствует напряжение на основном вводе ЩРПА
   |  *)

(* text list ClimateGroup (id | default)
  13 | Высокая температура
  12 | Низкая температура
  11 | Обогрев дверей выключен
  10 | Обогрев дверей включен
  9 | Кондиционеры выключены
  8 | Кондиционеры включены
  7 | Вентиляторы выключены
  6 | Вентиляторы включены
  5 | Заслонка закрыта
  4 | Заслонка открыта
  3 | Автоматика выключена
  2 | Обогрев выключен
  1 | Автоматика включена
  0 | Обогрев включен
   |  *)
